(* Logix 5000 project; controller pid Emulate 5570 rev 30.13; software revision 30.00 *)

TASK MainTask (continuous, watchdog 500 ms) : MainProgram

MODULES
   Local : Emulate 5570 (ICP 2, rev 30.13)
END_MODULES

VAR_GLOBAL   (* controller tags *)
   auto : BOOL := 1;
   auto_tune : PIDE_AUTOTUNE := (ProcessType := 3, ResponseSpeed := 1, PVTuneLimit := 10.0, StepSize := 10.0, TunedGood := 1, ATuneAcquired := 1, UsedProcessType := 6, Gain := 0.25000188, TimeConstant := 11.805334, DeadTime := 0.48400003, PGainTunedFast := 0.27980626, IGainTunedFast := 0.28487703, DGainTunedFast := 0.01070623, PGainTunedMed := 0.16587383, IGainTunedMed := 0.10388757, DGainTunedMed := 0.0064789923, PGainTunedSlow := 0.09402797, IGainTunedSlow := 0.03420702, DGainTunedSlow := 0.0037229029, StepSizeUsed := 10.0);
   bit1 : BOOL := 1;
   bit2 : BOOL := 1;
   Cal : BOOL;
   dd : COUNTER;
   float : REAL := 1.0425385;
   outon : BOOL := 1;
   outon1 : BOOL := 1;
   pid : PID := (CTL := -2147483648, EN := 1, SP := 40.0, MAXS := 4095.0, MAXO := 100.0, PV := 39.19998, MAXI := 4095.0, MAXCV := 100.0, MAXTIE := 100.0, DATA[4] := 40.0, DATA[5] := 0.024420025, DATA[6] := 1.0, DATA[15] := 1.0, DATA[16] := 1.0);
   PIDE_01 : PID_ENHANCED := (PV := 39.19998, PVEUMax := 80.0, SPProg := 40.0, SPOper := 40.0, SPHLimit := 80.0, RatioProg := 1.0, RatioOper := 1.0, RatioHLimit := 1.0, RatioLLimit := 1.0, CVEUMax := 100.0, CVHLimit := 100.0, PGain := 0.16587383, IGain := 0.10388757, DGain := 0.0064789923, PVEDerivative := 1, ProgProgReq := 1, ProgAutoReq := 1, RTSTime := 1, CVLAlarm := 1, SP := 40.0, SPPercent := 50.0, PVPercent := 48.999977, E := 0.8000183, EPercent := 1.0000229, InitPrimary := 1, WindupLOut := 1, Ratio := 1.0, ProgOper := 1, Auto := 1, DeltaT := 0.022000002, AtuneReady := 1, AtuneDone := 1);
   pv : REAL := 39.19998;
   shift : TIMER := (PRE := 25000, ACC := 12776, EN := 1, TT := 1);
   Sp : REAL := 40.0;
   t1 : TIMER := (PRE := 500, ACC := 519, EN := 1, DN := 1);
   up : COUNTER := (PRE := 10, ACC := 5);
END_VAR

PROGRAM MainProgram   (* main routine MainRoutine *)
VAR
   BNOT_01 : FBD_BOOLEAN_NOT := (In := 1);
END_VAR

ROUTINE MainRoutine   (* ladder *)
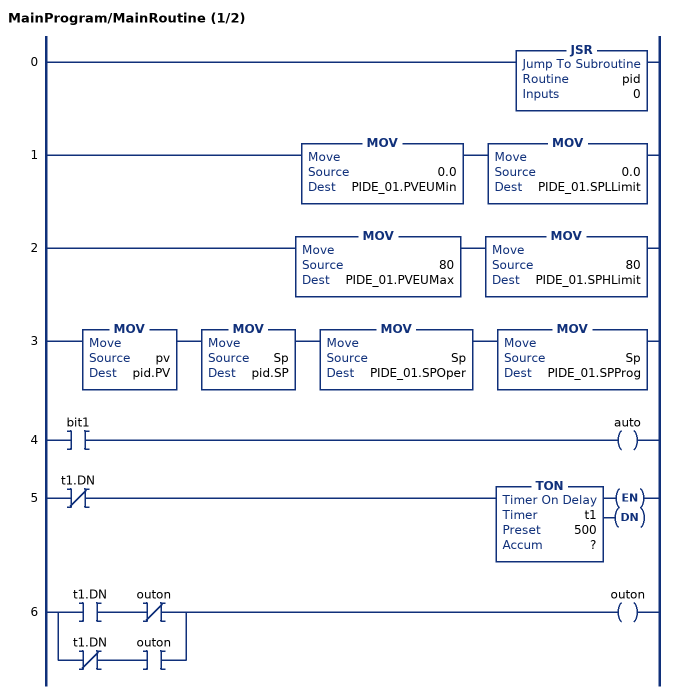
   0: JSR(pid,0);
   1: MOV(0.0,PIDE_01.PVEUMin)MOV(0.0,PIDE_01.SPLLimit);
   2: MOV(80,PIDE_01.PVEUMax)MOV(80,PIDE_01.SPHLimit);
   3: MOV(pv,pid.PV)MOV(Sp,pid.SP)MOV(Sp,PIDE_01.SPOper)MOV(Sp,PIDE_01.SPProg);
   4: XIC(bit1)OTE(auto);
   5: XIO(t1.DN)TON(t1,?,?);
   6: [XIC(t1.DN) XIO(outon) ,XIO(t1.DN) XIC(outon) ]OTE(outon);
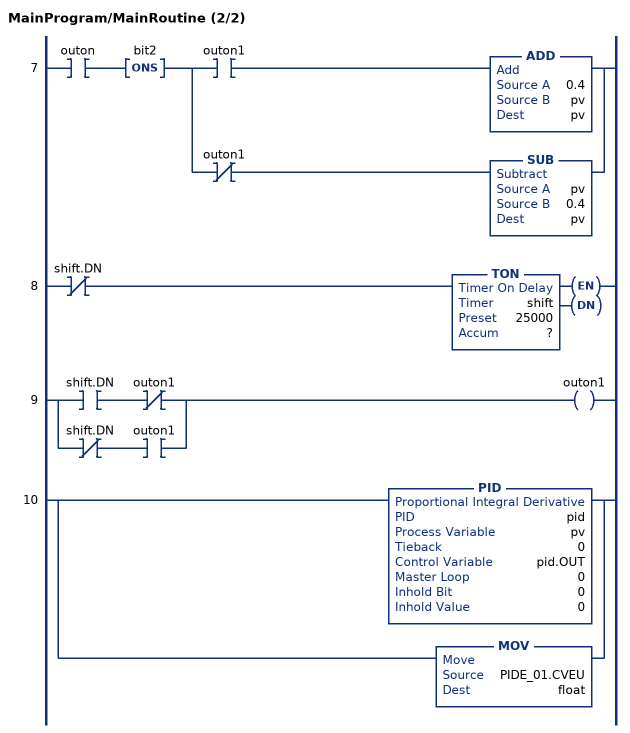
   7: XIC(outon)ONS(bit2)[XIC(outon1) ADD(0.4,pv,pv) ,XIO(outon1) SUB(pv,0.4,pv) ];
   8: XIO(shift.DN)TON(shift,?,?);
   9: [XIC(shift.DN) XIO(outon1) ,XIO(shift.DN) XIC(outon1) ]OTE(outon1);
   10: [PID(pid,pv,0,pid.OUT,0,0,0) ,MOV(PIDE_01.CVEU,float) ];
END_ROUTINE

ROUTINE pid   (* function block diagram *)
   SHEET 1
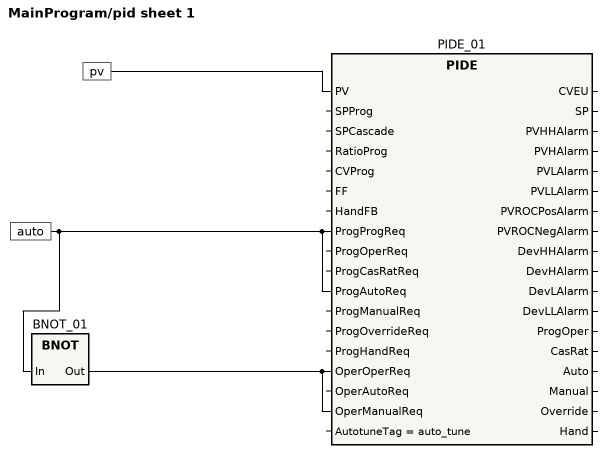
   BNOT_01 : BNOT(In := auto);
   PIDE_01 : PIDE(PV := pv, ProgProgReq := auto, ProgAutoReq := auto, OperOperReq := BNOT_01.Out, OperManualReq := BNOT_01.Out, AutotuneTag := auto_tune);   // unwired pins: SPProg SPCascade RatioProg CVProg FF HandFB ProgOperReq ProgCasRatReq ProgManualReq ProgOverrideReq ProgHandReq OperAutoReq CVEU SP PVHHAlarm PVHAlarm PVLAlarm PVLLAlarm PVROCPosAlarm PVROCNegAlarm DevHHAlarm DevHAlarm DevLAlarm DevLLAlarm ProgOper CasRat Auto Manual Override Hand
END_ROUTINE
END_PROGRAM
